LIN {X 0,Y 122.941,Z 954.134,A -85,B 0,C 180,E1 4520.76,E2 4520.76} C_VEL
LIN {X 0,Y 141.024,Z 945.626,A -85,B 0,C 180,E1 4515.408,E2 4515.408} C_VEL
LIN {X 0,Y 161.017,Z 934.73,A -85,B 0,C 180,E1 4511.199,E2 4511.199} C_VEL
LIN {X 0,Y 168.898,Z 929.93,A -85,B 0,C 180,E1 4509.837,E2 4509.837} C_VEL
LIN {X 0,Y 150.215,Z 939.451,A -85,B 0,C 180,E1 4506.112,E2 4506.112} C_VEL
LIN {X 0,Y 131.987,Z 947.261,A -85,B 0,C 180,E1 4501.242,E2 4501.242} C_VEL
LIN {X 0,Y 114.457,Z 953.373,A -85,B 0,C 180,E1 4494.654,E2 4494.654} C_VEL
LIN {X 0,Y 98.928,Z 957.725,A -85,B 0,C 180,E1 4485.934,E2 4485.934} C_VEL
LIN {X 0,Y 85.607,Z 960.518,A -85,B 0,C 180,E1 4473.649,E2 4473.649} C_VEL
LIN {X 0,Y 77.458,Z 961.489,A -85,B 0,C 180,E1 4459.579,E2 4459.579} C_VEL
LIN {X 0,Y 73.991,Z 961.027,A -85,B 0,C 180,E1 4445.504,E2 4445.504} C_VEL
LIN {X 0,Y 73.516,Z 959.727,A -85,B 0,C 180,E1 4432.349,E2 4432.349} C_VEL
LIN {X 0,Y 75.609,Z 957.116,A -85,B 0,C 180,E1 4418.348,E2 4418.348} C_VEL
LIN {X 0,Y 81.937,Z 952.659,A -85,B 0,C 180,E1 4403.68,E2 4403.68} C_VEL
LIN {X 0,Y 91.415,Z 946.902,A -85,B 0,C 180,E1 4392.153,E2 4392.153} C_VEL
LIN {X 0,Y 104.12,Z 938.983,A -85,B 0,C 180,E1 4382.54,E2 4382.54} C_VEL
LIN {X 0,Y 118.028,Z 929.614,A -85,B 0,C 180,E1 4375.407,E2 4375.407} C_VEL
LIN {X 0,Y 133.192,Z 918.259,A -85,B 0,C 180,E1 4369.779,E2 4369.779} C_VEL
LIN {X 0,Y 148.363,Z 905.384,A -85,B 0,C 180,E1 4365.492,E2 4365.492} C_VEL
LIN {X 0,Y 162.344,Z 891.921,A -85,B 0,C 180,E1 4362.339,E2 4362.339} C_VEL
LIN {X 0,Y 176.658,Z 876.08,A -85,B 0,C 180,E1 4359.661,E2 4359.661} C_VEL
LIN {X 0,Y 189.851,Z 859.095,A -85,B 0,C 180,E1 4357.561,E2 4357.561} C_VEL
LIN {X 0,Y 201.371,Z 841.861,A -85,B 0,C 180,E1 4355.961,E2 4355.961} C_VEL
LIN {X 0,Y 212.517,Z 822.257,A -85,B 0,C 180,E1 4354.571,E2 4354.571} C_VEL
LIN {X 0,Y 221.857,Z 802.538,A -85,B 0,C 180,E1 4353.507,E2 4353.507} C_VEL
LIN {X 0,Y 229.677,Z 782.335,A -85,B 0,C 180,E1 4352.672,E2 4352.672} C_VEL
LIN {X 0,Y 236.26,Z 760.464,A -85,B 0,C 180,E1 4351.999,E2 4351.999} C_VEL
LIN {X 0,Y 241.017,Z 738.583,A -85,B 0,C 180,E1 4351.512,E2 4351.512} C_VEL
LIN {X 0,Y 245.764,Z 704.393,A -85,B 0,C 180,E1 4350.967,E2 4350.967} C_VEL
LIN {X 0,Y 252.811,Z 648.458,A -85,B 0,C 180,E1 4350.086,E2 4350.086} C_VEL
LIN {X 0,Y 251.155,Z 644.335,A -85,B 0,C 180,E1 4346.898,E2 4346.898} C_VEL
LIN {X 0,Y 250.174,Z 641.772,A -85,B 0,C 180,E1 4344.31,E2 4344.31} C_VEL
LIN {X 0,Y 249.238,Z 639.151,A -85,B 0,C 180,E1 4340.152,E2 4340.152} C_VEL
LIN {X 0,Y 249.155,Z 638.957,A -85,B 0,C 180,E1 4334.645,E2 4334.645} C_VEL
LIN {X 0,Y 249.526,Z 639.799,A -85,B 0,C 180,E1 4332.262,E2 4332.262} C_VEL
LIN {X 0,Y 250.94,Z 643.145,A -85,B 0,C 180,E1 4327.787,E2 4327.787} C_VEL
LIN {X 0,Y 252.591,Z 647.143,A -85,B 0,C 180,E1 4324.428,E2 4324.428} C_VEL
LIN {X 0,Y 254.618,Z 652.06,A -85,B 0,C 180,E1 4321.288,E2 4321.288} C_VEL
LIN {X 0,Y 243.355,Z 742.447,A -85,B 0,C 180,E1 4319.848,E2 4319.848} C_VEL
LIN {X 0,Y 238.68,Z 764.766,A -85,B 0,C 180,E1 4319.412,E2 4319.412} C_VEL
LIN {X 0,Y 232.693,Z 785.189,A -85,B 0,C 180,E1 4318.95,E2 4318.95} C_VEL
LIN {X 0,Y 224.583,Z 806.826,A -85,B 0,C 180,E1 4318.285,E2 4318.285} C_VEL
LIN {X 0,Y 215.694,Z 826.159,A -85,B 0,C 180,E1 4317.468,E2 4317.468} C_VEL
LIN {X 0,Y 205.01,Z 845.556,A -85,B 0,C 180,E1 4316.366,E2 4316.366} C_VEL
LIN {X 0,Y 192.977,Z 863.966,A -85,B 0,C 180,E1 4314.948,E2 4314.948} C_VEL
LIN {X 0,Y 180.253,Z 880.755,A -85,B 0,C 180,E1 4313.213,E2 4313.213} C_VEL
LIN {X 0,Y 166.08,Z 897.05,A -85,B 0,C 180,E1 4310.907,E2 4310.907} C_VEL
LIN {X 0,Y 151.319,Z 911.904,A -85,B 0,C 180,E1 4307.969,E2 4307.969} C_VEL
LIN {X 0,Y 136.169,Z 925.263,A -85,B 0,C 180,E1 4304.161,E2 4304.161} C_VEL
LIN {X 0,Y 133.634,Z 927.346,A -85,B 0,C 180,E1 4303.421,E2 4303.421} C_VEL
LIN {X 0,Y 127.746,Z 931.563,A -85,B 0,C 180,E1 4302.123,E2 4302.123} C_VEL
LIN {X 0,Y 110.847,Z 941.115,A -85,B 0,C 180,E1 4299.58,E2 4299.58} C_VEL
LIN {X 0,Y 104.946,Z 944.656,A -85,B 0,C 180,E1 4297.699,E2 4297.699} C_VEL
LIN {X 0,Y 90.296,Z 953.759,A -85,B 0,C 180,E1 4289.381,E2 4289.381} C_VEL
LIN {X 0,Y 77.912,Z 961.092,A -85,B 0,C 180,E1 4278.122,E2 4278.122} C_VEL
LIN {X 0,Y 69.097,Z 966.731,A -85,B 0,C 180,E1 4263.378,E2 4263.378} C_VEL
LIN {X 0,Y 65.327,Z 970.268,A -85,B 0,C 180,E1 4247.844,E2 4247.844} C_VEL
LIN {X 0,Y 65.237,Z 972.242,A -85,B 0,C 180,E1 4233.533,E2 4233.533} C_VEL
LIN {X 0,Y 65.26,Z 972.617,A -85,B 0,C 180,E1 4227.384,E2 4227.384} C_VEL
LIN {X 0,Y 65.112,Z 972.66,A -85,B 0,C 180,E1 4213.057,E2 4213.057} C_VEL
LIN {X 0,Y 69.713,Z 971.183,A -85,B 0,C 180,E1 4194.833,E2 4194.833} C_VEL
LIN {X 0,Y 80.755,Z 967.951,A -85,B 0,C 180,E1 4178.764,E2 4178.764} C_VEL
LIN {X 0,Y 97.243,Z 962.683,A -85,B 0,C 180,E1 4166.583,E2 4166.583} C_VEL
LIN {X 0,Y 116.788,Z 955.393,A -85,B 0,C 180,E1 4158.178,E2 4158.178} C_VEL
LIN {X 0,Y 136.489,Z 946.767,A -85,B 0,C 180,E1 4152.694,E2 4152.694} C_VEL
LIN {X 0,Y 151.098,Z 939.539,A -85,B 0,C 180,E1 4149.665,E2 4149.665} C_VEL
LIN {X 0,Y 131.493,Z 947.642,A -85,B 0,C 180,E1 4145.181,E2 4145.181} C_VEL
LIN {X 0,Y 112.97,Z 953.837,A -85,B 0,C 180,E1 4139.187,E2 4139.187} C_VEL
LIN {X 0,Y 96.095,Z 958.284,A -85,B 0,C 180,E1 4131.019,E2 4131.019} C_VEL
LIN {X 0,Y 81.927,Z 961.07,A -85,B 0,C 180,E1 4119.958,E2 4119.958} C_VEL
LIN {X 0,Y 71.187,Z 962.264,A -85,B 0,C 180,E1 4104.52,E2 4104.52} C_VEL
LIN {X 0,Y 66.324,Z 961.804,A -85,B 0,C 180,E1 4088.152,E2 4088.152} C_VEL
LIN {X 0,Y 65.487,Z 960.535,A -85,B 0,C 180,E1 4073.633,E2 4073.633} C_VEL
LIN {X 0,Y 67.428,Z 958.096,A -85,B 0,C 180,E1 4058.509,E2 4058.509} C_VEL
LIN {X 0,Y 73.652,Z 954.042,A -85,B 0,C 180,E1 4042.966,E2 4042.966} C_VEL
LIN {X 0,Y 84.182,Z 948.085,A -85,B 0,C 180,E1 4029.837,E2 4029.837} C_VEL
LIN {X 0,Y 96.897,Z 940.726,A -85,B 0,C 180,E1 4020.297,E2 4020.297} C_VEL
LIN {X 0,Y 112.186,Z 931.095,A -85,B 0,C 180,E1 4012.683,E2 4012.683} C_VEL
LIN {X 0,Y 127.924,Z 919.921,A -85,B 0,C 180,E1 4007.146,E2 4007.146} C_VEL
LIN {X 0,Y 142.681,Z 908.045,A -85,B 0,C 180,E1 4003.204,E2 4003.204} C_VEL
LIN {X 0,Y 157.899,Z 893.971,A -85,B 0,C 180,E1 3999.976,E2 3999.976} C_VEL
LIN {X 0,Y 172.065,Z 878.845,A -85,B 0,C 180,E1 3997.506,E2 3997.506} C_VEL
LIN {X 0,Y 185.501,Z 862.283,A -85,B 0,C 180,E1 3995.513,E2 3995.513} C_VEL
LIN {X 0,Y 198.155,Z 844.091,A -85,B 0,C 180,E1 3993.889,E2 3993.889} C_VEL
LIN {X 0,Y 209.006,Z 825.752,A -85,B 0,C 180,E1 3992.644,E2 3992.644} C_VEL
LIN {X 0,Y 218.958,Z 805.636,A -85,B 0,C 180,E1 3991.602,E2 3991.602} C_VEL
LIN {X 0,Y 227.293,Z 784.765,A -85,B 0,C 180,E1 3990.783,E2 3990.783} C_VEL
LIN {X 0,Y 233.847,Z 763.8,A -85,B 0,C 180,E1 3990.168,E2 3990.168} C_VEL
LIN {X 0,Y 238.893,Z 742.056,A -85,B 0,C 180,E1 3989.697,E2 3989.697} C_VEL
LIN {X 0,Y 243.144,Z 713.786,A -85,B 0,C 180,E1 3989.258,E2 3989.258} C_VEL
LIN {X 0,Y 250.728,Z 654.36,A -85,B 0,C 180,E1 3988.374,E2 3988.374} C_VEL
LIN {X 0,Y 249.208,Z 650.025,A -85,B 0,C 180,E1 3984.663,E2 3984.663} C_VEL
LIN {X 0,Y 248.14,Z 647.059,A -85,B 0,C 180,E1 3980.03,E2 3980.03} C_VEL
LIN {X 0,Y 248.104,Z 646.928,A -85,B 0,C 180,E1 3974.47,E2 3974.47} C_VEL
LIN {X 0,Y 248.426,Z 647.784,A -85,B 0,C 180,E1 3972.317,E2 3972.317} C_VEL
LIN {X 0,Y 249.675,Z 650.864,A -85,B 0,C 180,E1 3968.174,E2 3968.174} C_VEL
LIN {X 0,Y 251.255,Z 654.891,A -85,B 0,C 180,E1 3964.794,E2 3964.794} C_VEL
LIN {X 0,Y 252.333,Z 657.73,A -85,B 0,C 180,E1 3962.976,E2 3962.976} C_VEL
LIN {X 0,Y 241.585,Z 742.196,A -85,B 0,C 180,E1 3961.695,E2 3961.695} C_VEL
LIN {X 0,Y 236.821,Z 764.595,A -85,B 0,C 180,E1 3961.289,E2 3961.289} C_VEL
LIN {X 0,Y 230.507,Z 785.745,A -85,B 0,C 180,E1 3960.853,E2 3960.853} C_VEL
LIN {X 0,Y 222.409,Z 806.917,A -85,B 0,C 180,E1 3960.258,E2 3960.258} C_VEL
LIN {X 0,Y 212.993,Z 826.926,A -85,B 0,C 180,E1 3959.48,E2 3959.48} C_VEL
LIN {X 0,Y 202.059,Z 846.323,A -85,B 0,C 180,E1 3958.458,E2 3958.458} C_VEL
LIN {X 0,Y 189.725,Z 864.773,A -85,B 0,C 180,E1 3957.137,E2 3957.137} C_VEL
LIN {X 0,Y 176.536,Z 881.669,A -85,B 0,C 180,E1 3955.496,E2 3955.496} C_VEL
LIN {X 0,Y 162.089,Z 897.747,A -85,B 0,C 180,E1 3953.335,E2 3953.335} C_VEL
LIN {X 0,Y 146.987,Z 912.405,A -85,B 0,C 180,E1 3950.56,E2 3950.56} C_VEL
LIN {X 0,Y 131.407,Z 925.655,A -85,B 0,C 180,E1 3946.923,E2 3946.923} C_VEL
LIN {X 0,Y 115.629,Z 937.38,A -85,B 0,C 180,E1 3942.052,E2 3942.052} C_VEL
LIN {X 0,Y 104.946,Z 944.656,A -85,B 0,C 180,E1 3937.699,E2 3937.699} C_VEL
LIN {X 0,Y 99.077,Z 948.011,A -85,B 0,C 180,E1 3935.556,E2 3935.556} C_VEL
LIN {X 0,Y 81.245,Z 955.584,A -85,B 0,C 180,E1 3929.929,E2 3929.929} C_VEL
LIN {X 0,Y 76.561,Z 957.802,A -85,B 0,C 180,E1 3926.89,E2 3926.89} C_VEL
LIN {X 0,Y 65.424,Z 963.843,A -85,B 0,C 180,E1 3913.474,E2 3913.474} C_VEL
LIN {X 0,Y 58.448,Z 968.456,A -85,B 0,C 180,E1 3895.342,E2 3895.342} C_VEL
LIN {X 0,Y 57.026,Z 970.951,A -85,B 0,C 180,E1 3878.085,E2 3878.085} C_VEL
LIN {X 0,Y 57.431,Z 971.671,A -85,B 0,C 180,E1 3870.021,E2 3870.021} C_VEL
LIN {X 0,Y 56.913,Z 971.987,A -85,B 0,C 180,E1 3857.852,E2 3857.852} C_VEL
LIN {X 0,Y 60.005,Z 971.266,A -85,B 0,C 180,E1 3838.185,E2 3838.185} C_VEL
LIN {X 0,Y 70.752,Z 968.681,A -85,B 0,C 180,E1 3819.02,E2 3819.02} C_VEL
LIN {X 0,Y 86.659,Z 964.409,A -85,B 0,C 180,E1 3805.884,E2 3805.884} C_VEL
LIN {X 0,Y 105.789,Z 958.337,A -85,B 0,C 180,E1 3797.036,E2 3797.036} C_VEL
LIN {X 0,Y 126.327,Z 950.451,A -85,B 0,C 180,E1 3791.115,E2 3791.115} C_VEL
LIN {X 0,Y 133.3,Z 947.425,A -85,B 0,C 180,E1 3789.497,E2 3789.497} C_VEL
LIN {X 0,Y 112.982,Z 954.102,A -85,B 0,C 180,E1 3784.058,E2 3784.058} C_VEL
LIN {X 0,Y 94.015,Z 958.884,A -85,B 0,C 180,E1 3776.34,E2 3776.34} C_VEL
LIN {X 0,Y 77.524,Z 961.836,A -85,B 0,C 180,E1 3765.241,E2 3765.241} C_VEL
LIN {X 0,Y 65.004,Z 963.029,A -85,B 0,C 180,E1 3749.43,E2 3749.43} C_VEL
LIN {X 0,Y 58.82,Z 962.581,A -85,B 0,C 180,E1 3731.496,E2 3731.496} C_VEL
LIN {X 0,Y 57.477,Z 961.326,A -85,B 0,C 180,E1 3715.225,E2 3715.225} C_VEL
LIN {X 0,Y 59.506,Z 958.849,A -85,B 0,C 180,E1 3697.52,E2 3697.52} C_VEL
LIN {X 0,Y 66.296,Z 954.862,A -85,B 0,C 180,E1 3680.432,E2 3680.432} C_VEL
LIN {X 0,Y 77.764,Z 948.921,A -85,B 0,C 180,E1 3666.494,E2 3666.494} C_VEL
LIN {X 0,Y 91.366,Z 941.604,A -85,B 0,C 180,E1 3656.812,E2 3656.812} C_VEL
LIN {X 0,Y 107.459,Z 932.02,A -85,B 0,C 180,E1 3649.345,E2 3649.345} C_VEL
LIN {X 0,Y 123.463,Z 921.171,A -85,B 0,C 180,E1 3644.146,E2 3644.146} C_VEL
LIN {X 0,Y 139.051,Z 909.084,A -85,B 0,C 180,E1 3640.33,E2 3640.33} C_VEL
LIN {X 0,Y 154.659,Z 895.043,A -85,B 0,C 180,E1 3637.317,E2 3637.317} C_VEL
LIN {X 0,Y 168.722,Z 880.448,A -85,B 0,C 180,E1 3635.089,E2 3635.089} C_VEL
LIN {X 0,Y 182.82,Z 863.531,A -85,B 0,C 180,E1 3633.19,E2 3633.19} C_VEL
LIN {X 0,Y 195.204,Z 846.205,A -85,B 0,C 180,E1 3631.75,E2 3631.75} C_VEL
LIN {X 0,Y 206.692,Z 827.288,A -85,B 0,C 180,E1 3630.555,E2 3630.555} C_VEL
LIN {X 0,Y 216.775,Z 807.316,A -85,B 0,C 180,E1 3629.598,E2 3629.598} C_VEL
LIN {X 0,Y 224.941,Z 787.416,A -85,B 0,C 180,E1 3628.869,E2 3628.869} C_VEL
LIN {X 0,Y 231.868,Z 766.149,A -85,B 0,C 180,E1 3628.28,E2 3628.28} C_VEL
LIN {X 0,Y 237.323,Z 743.515,A -85,B 0,C 180,E1 3627.821,E2 3627.821} C_VEL
LIN {X 0,Y 241.195,Z 719.145,A -85,B 0,C 180,E1 3627.462,E2 3627.462} C_VEL
LIN {X 0,Y 248.821,Z 660.307,A -85,B 0,C 180,E1 3626.652,E2 3626.652} C_VEL
LIN {X 0,Y 247.741,Z 657.272,A -85,B 0,C 180,E1 3623.551,E2 3623.551} C_VEL
LIN {X 0,Y 247.039,Z 654.961,A -85,B 0,C 180,E1 3619.876,E2 3619.876} C_VEL
LIN {X 0,Y 247.02,Z 654.849,A -85,B 0,C 180,E1 3614.535,E2 3614.535} C_VEL
LIN {X 0,Y 247.327,Z 655.766,A -85,B 0,C 180,E1 3612.373,E2 3612.373} C_VEL
LIN {X 0,Y 248.463,Z 658.715,A -85,B 0,C 180,E1 3608.447,E2 3608.447} C_VEL
LIN {X 0,Y 249.966,Z 662.73,A -85,B 0,C 180,E1 3605.096,E2 3605.096} C_VEL
LIN {X 0,Y 250.168,Z 663.427,A -85,B 0,C 180,E1 3604.689,E2 3604.689} C_VEL
LIN {X 0,Y 240.027,Z 741.859,A -85,B 0,C 180,E1 3603.566,E2 3603.566} C_VEL
LIN {X 0,Y 235.208,Z 764.284,A -85,B 0,C 180,E1 3603.192,E2 3603.192} C_VEL
LIN {X 0,Y 228.755,Z 785.662,A -85,B 0,C 180,E1 3602.801,E2 3602.801} C_VEL
LIN {X 0,Y 220.844,Z 806.154,A -85,B 0,C 180,E1 3602.292,E2 3602.292} C_VEL
LIN {X 0,Y 211.644,Z 825.647,A -85,B 0,C 180,E1 3601.625,E2 3601.625} C_VEL
LIN {X 0,Y 200.502,Z 845.307,A -85,B 0,C 180,E1 3600.708,E2 3600.708} C_VEL
LIN {X 0,Y 187.995,Z 863.798,A -85,B 0,C 180,E1 3599.526,E2 3599.526} C_VEL
LIN {X 0,Y 175.086,Z 880.175,A -85,B 0,C 180,E1 3598.107,E2 3598.107} C_VEL
LIN {X 0,Y 160.352,Z 896.398,A -85,B 0,C 180,E1 3596.167,E2 3596.167} C_VEL
LIN {X 0,Y 145.842,Z 910.358,A -85,B 0,C 180,E1 3593.827,E2 3593.827} C_VEL
LIN {X 0,Y 129.76,Z 923.761,A -85,B 0,C 180,E1 3590.551,E2 3590.551} C_VEL
LIN {X 0,Y 113.948,Z 935.294,A -85,B 0,C 180,E1 3586.297,E2 3586.297} C_VEL
LIN {X 0,Y 96.937,Z 946.232,A -85,B 0,C 180,E1 3579.853,E2 3579.853} C_VEL
LIN {X 0,Y 82.081,Z 954.798,A -85,B 0,C 180,E1 3571.317,E2 3571.317} C_VEL
LIN {X 0,Y 76.561,Z 957.802,A -85,B 0,C 180,E1 3566.89,E2 3566.89} C_VEL
LIN {X 0,Y 71.268,Z 960.225,A -85,B 0,C 180,E1 3562.908,E2 3562.908} C_VEL
LIN {X 0,Y 55.416,Z 965.293,A -85,B 0,C 180,E1 3549.962,E2 3549.962} C_VEL
LIN {X 0,Y 52.571,Z 966.514,A -85,B 0,C 180,E1 3544.351,E2 3544.351} C_VEL
LIN {X 0,Y 49.05,Z 969.709,A -85,B 0,C 180,E1 3522.983,E2 3522.983} C_VEL
LIN {X 0,Y 49.46,Z 970.859,A -85,B 0,C 180,E1 3510.025,E2 3510.025} C_VEL
LIN {X 0,Y 49.106,Z 971.19,A -85,B 0,C 180,E1 3493.464,E2 3493.464} C_VEL
LIN {X 0,Y 54.103,Z 970.401,A -85,B 0,C 180,E1 3471.103,E2 3471.103} C_VEL
LIN {X 0,Y 67.203,Z 967.806,A -85,B 0,C 180,E1 3452.036,E2 3452.036} C_VEL
LIN {X 0,Y 85.869,Z 963.286,A -85,B 0,C 180,E1 3439.458,E2 3439.458} C_VEL
LIN {X 0,Y 106.229,Z 957.201,A -85,B 0,C 180,E1 3431.863,E2 3431.863} C_VEL
LIN {X 0,Y 115.656,Z 953.892,A -85,B 0,C 180,E1 3429.36,E2 3429.36} C_VEL
LIN {X 0,Y 95.075,Z 959.065,A -85,B 0,C 180,E1 3422.787,E2 3422.787} C_VEL
LIN {X 0,Y 76.527,Z 962.262,A -85,B 0,C 180,E1 3413.055,E2 3413.055} C_VEL
LIN {X 0,Y 62.013,Z 963.646,A -85,B 0,C 180,E1 3399.193,E2 3399.193} C_VEL
LIN {X 0,Y 52.173,Z 963.481,A -85,B 0,C 180,E1 3378.329,E2 3378.329} C_VEL
LIN {X 0,Y 49.565,Z 962.31,A -85,B 0,C 180,E1 3359.833,E2 3359.833} C_VEL
LIN {X 0,Y 50.826,Z 960.22,A -85,B 0,C 180,E1 3340.173,E2 3340.173} C_VEL
LIN {X 0,Y 57.078,Z 956.585,A -85,B 0,C 180,E1 3320.908,E2 3320.908} C_VEL
LIN {X 0,Y 68.867,Z 951.03,A -85,B 0,C 180,E1 3305.081,E2 3305.081} C_VEL
LIN {X 0,Y 82.999,Z 944.158,A -85,B 0,C 180,E1 3294.657,E2 3294.657} C_VEL
LIN {X 0,Y 98.79,Z 935.543,A -85,B 0,C 180,E1 3287.289,E2 3287.289} C_VEL
LIN {X 0,Y 114.757,Z 925.504,A -85,B 0,C 180,E1 3282.138,E2 3282.138} C_VEL
LIN {X 0,Y 131.136,Z 913.677,A -85,B 0,C 180,E1 3278.236,E2 3278.236} C_VEL
LIN {X 0,Y 147.132,Z 900.325,A -85,B 0,C 180,E1 3275.285,E2 3275.285} C_VEL
LIN {X 0,Y 162.227,Z 885.765,A -85,B 0,C 180,E1 3273.037,E2 3273.037} C_VEL
LIN {X 0,Y 176.604,Z 869.569,A -85,B 0,C 180,E1 3271.241,E2 3271.241} C_VEL
LIN {X 0,Y 189.542,Z 852.545,A -85,B 0,C 180,E1 3269.844,E2 3269.844} C_VEL
LIN {X 0,Y 201.74,Z 833.693,A -85,B 0,C 180,E1 3268.679,E2 3268.679} C_VEL
LIN {X 0,Y 212.427,Z 813.966,A -85,B 0,C 180,E1 3267.754,E2 3267.754} C_VEL
LIN {X 0,Y 221.179,Z 794.421,A -85,B 0,C 180,E1 3267.049,E2 3267.049} C_VEL
LIN {X 0,Y 228.712,Z 773.36,A -85,B 0,C 180,E1 3266.47,E2 3266.47} C_VEL
LIN {X 0,Y 234.617,Z 751.43,A -85,B 0,C 180,E1 3266.024,E2 3266.024} C_VEL
LIN {X 0,Y 238.698,Z 729.638,A -85,B 0,C 180,E1 3265.704,E2 3265.704} C_VEL
LIN {X 0,Y 247.05,Z 666.591,A -85,B 0,C 180,E1 3264.893,E2 3264.893} C_VEL
LIN {X 0,Y 246.332,Z 664.418,A -85,B 0,C 180,E1 3262.255,E2 3262.255} C_VEL
LIN {X 0,Y 245.91,Z 662.815,A -85,B 0,C 180,E1 3259.476,E2 3259.476} C_VEL
LIN {X 0,Y 245.969,Z 662.824,A -85,B 0,C 180,E1 3254.358,E2 3254.358} C_VEL
LIN {X 0,Y 246.325,Z 664.07,A -85,B 0,C 180,E1 3251.948,E2 3251.948} C_VEL
LIN {X 0,Y 247.259,Z 666.566,A -85,B 0,C 180,E1 3248.723,E2 3248.723} C_VEL
LIN {X 0,Y 248.197,Z 669.297,A -85,B 0,C 180,E1 3246.428,E2 3246.428} C_VEL
LIN {X 0,Y 238.688,Z 741.456,A -85,B 0,C 180,E1 3245.459,E2 3245.459} C_VEL
LIN {X 0,Y 233.814,Z 763.887,A -85,B 0,C 180,E1 3245.119,E2 3245.119} C_VEL
LIN {X 0,Y 227.322,Z 785.215,A -85,B 0,C 180,E1 3244.78,E2 3244.78} C_VEL
LIN {X 0,Y 219.108,Z 806.245,A -85,B 0,C 180,E1 3244.326,E2 3244.326} C_VEL
LIN {X 0,Y 209.425,Z 826.352,A -85,B 0,C 180,E1 3243.717,E2 3243.717} C_VEL
LIN {X 0,Y 198.243,Z 845.688,A -85,B 0,C 180,E1 3242.914,E2 3242.914} C_VEL
LIN {X 0,Y 185.468,Z 864.286,A -85,B 0,C 180,E1 3241.855,E2 3241.855} C_VEL
LIN {X 0,Y 171.999,Z 880.964,A -85,B 0,C 180,E1 3240.551,E2 3240.551} C_VEL
LIN {X 0,Y 157.028,Z 896.988,A -85,B 0,C 180,E1 3238.801,E2 3238.801} C_VEL
LIN {X 0,Y 141.258,Z 911.595,A -85,B 0,C 180,E1 3236.518,E2 3236.518} C_VEL
LIN {X 0,Y 124.811,Z 924.796,A -85,B 0,C 180,E1 3233.466,E2 3233.466} C_VEL
LIN {X 0,Y 106.973,Z 937.101,A -85,B 0,C 180,E1 3228.987,E2 3228.987} C_VEL
LIN {X 0,Y 90.887,Z 946.713,A -85,B 0,C 180,E1 3223.197,E2 3223.197} C_VEL
LIN {X 0,Y 74.511,Z 955.408,A -85,B 0,C 180,E1 3214.07,E2 3214.07} C_VEL
LIN {X 0,Y 60.823,Z 962.168,A -85,B 0,C 180,E1 3200.619,E2 3200.619} C_VEL
LIN {X 0,Y 52.571,Z 966.514,A -85,B 0,C 180,E1 3184.351,E2 3184.351} C_VEL
LIN {X 0,Y 49.652,Z 967.94,A -85,B 0,C 180,E1 3176.39,E2 3176.39} C_VEL
LIN {X 0,Y 45.336,Z 969.237,A -85,B 0,C 180,E1 3164.722,E2 3164.722} C_VEL
LIN {X 0,Y 41.036,Z 970.251,A -85,B 0,C 180,E1 3141.827,E2 3141.827} C_VEL
LIN {X 0,Y 44.01,Z 970.224,A -85,B 0,C 180,E1 3115.426,E2 3115.426} C_VEL
LIN {X 0,Y 56.367,Z 968.429,A -85,B 0,C 180,E1 3092.147,E2 3092.147} C_VEL
LIN {X 0,Y 75.529,Z 964.711,A -85,B 0,C 180,E1 3077.668,E2 3077.668} C_VEL
LIN {X 0,Y 97.263,Z 959.178,A -85,B 0,C 180,E1 3069.381,E2 3069.381} C_VEL
LIN {X 0,Y 97.673,Z 959.038,A -85,B 0,C 180,E1 3069.134,E2 3069.134} C_VEL
LIN {X 0,Y 77.99,Z 962.496,A -85,B 0,C 180,E1 3061.456,E2 3061.456} C_VEL
LIN {X 0,Y 60.106,Z 964.319,A -85,B 0,C 180,E1 3048.836,E2 3048.836} C_VEL
LIN {X 0,Y 46.928,Z 964.45,A -85,B 0,C 180,E1 3028.405,E2 3028.405} C_VEL
LIN {X 0,Y 41.863,Z 963.217,A -85,B 0,C 180,E1 3004.938,E2 3004.938} C_VEL
LIN {X 0,Y 42.053,Z 961.569,A -85,B 0,C 180,E1 2985.131,E2 2985.131} C_VEL
LIN {X 0,Y 47.821,Z 958.273,A -85,B 0,C 180,E1 2961.559,E2 2961.559} C_VEL
LIN {X 0,Y 59.3,Z 953.426,A -85,B 0,C 180,E1 2943.977,E2 2943.977} C_VEL
LIN {X 0,Y 74.981,Z 946.454,A -85,B 0,C 180,E1 2931.886,E2 2931.886} C_VEL
LIN {X 0,Y 91.554,Z 938.084,A -85,B 0,C 180,E1 2924.345,E2 2924.345} C_VEL
LIN {X 0,Y 109.353,Z 927.631,A -85,B 0,C 180,E1 2918.981,E2 2918.981} C_VEL
LIN {X 0,Y 126.252,Z 916.05,A -85,B 0,C 180,E1 2915.328,E2 2915.328} C_VEL
LIN {X 0,Y 142.494,Z 903.111,A -85,B 0,C 180,E1 2912.633,E2 2912.633} C_VEL
LIN {X 0,Y 157.945,Z 888.703,A -85,B 0,C 180,E1 2910.566,E2 2910.566} C_VEL
LIN {X 0,Y 172.538,Z 872.912,A -85,B 0,C 180,E1 2908.938,E2 2908.938} C_VEL
LIN {X 0,Y 186.712,Z 854.951,A -85,B 0,C 180,E1 2907.582,E2 2907.582} C_VEL
LIN {X 0,Y 198.976,Z 836.61,A -85,B 0,C 180,E1 2906.551,E2 2906.551} C_VEL
LIN {X 0,Y 209.783,Z 817.41,A -85,B 0,C 180,E1 2905.726,E2 2905.726} C_VEL
LIN {X 0,Y 219.116,Z 797.237,A -85,B 0,C 180,E1 2905.061,E2 2905.061} C_VEL
LIN {X 0,Y 226.721,Z 776.656,A -85,B 0,C 180,E1 2904.544,E2 2904.544} C_VEL
LIN {X 0,Y 232.87,Z 755.049,A -85,B 0,C 180,E1 2904.134,E2 2904.134} C_VEL
LIN {X 0,Y 237.489,Z 731.912,A -85,B 0,C 180,E1 2903.817,E2 2903.817} C_VEL
LIN {X 0,Y 245.425,Z 672.981,A -85,B 0,C 180,E1 2903.087,E2 2903.087} C_VEL
LIN {X 0,Y 244.815,Z 670.719,A -85,B 0,C 180,E1 2899.319,E2 2899.319} C_VEL
LIN {X 0,Y 244.915,Z 670.798,A -85,B 0,C 180,E1 2894.179,E2 2894.179} C_VEL
LIN {X 0,Y 245.954,Z 674.02,A -85,B 0,C 180,E1 2889.359,E2 2889.359} C_VEL
LIN {X 0,Y 246.326,Z 675.457,A -85,B 0,C 180,E1 2888.187,E2 2888.187} C_VEL
LIN {X 0,Y 237.52,Z 741.248,A -85,B 0,C 180,E1 2887.366,E2 2887.366} C_VEL
LIN {X 0,Y 232.622,Z 763.586,A -85,B 0,C 180,E1 2887.064,E2 2887.064} C_VEL
LIN {X 0,Y 226.27,Z 784.353,A -85,B 0,C 180,E1 2886.786,E2 2886.786} C_VEL
LIN {X 0,Y 218.355,Z 804.674,A -85,B 0,C 180,E1 2886.425,E2 2886.425} C_VEL
LIN {X 0,Y 209.109,Z 824.072,A -85,B 0,C 180,E1 2885.943,E2 2885.943} C_VEL
LIN {X 0,Y 197.822,Z 843.695,A -85,B 0,C 180,E1 2885.267,E2 2885.267} C_VEL
LIN {X 0,Y 185.541,Z 861.582,A -85,B 0,C 180,E1 2884.419,E2 2884.419} C_VEL
LIN {X 0,Y 172.094,Z 878.388,A -85,B 0,C 180,E1 2883.332,E2 2883.332} C_VEL
LIN {X 0,Y 157.078,Z 894.547,A -85,B 0,C 180,E1 2881.874,E2 2881.874} C_VEL
LIN {X 0,Y 141.475,Z 909.058,A -85,B 0,C 180,E1 2880.001,E2 2880.001} C_VEL
LIN {X 0,Y 125.118,Z 922.093,A -85,B 0,C 180,E1 2877.508,E2 2877.508} C_VEL
LIN {X 0,Y 108.566,Z 933.528,A -85,B 0,C 180,E1 2874.16,E2 2874.16} C_VEL
LIN {X 0,Y 91.327,Z 943.859,A -85,B 0,C 180,E1 2869.275,E2 2869.275} C_VEL
LIN {X 0,Y 74.535,Z 952.576,A -85,B 0,C 180,E1 2862.031,E2 2862.031} C_VEL
LIN {X 0,Y 58.725,Z 959.756,A -85,B 0,C 180,E1 2850.305,E2 2850.305} C_VEL
LIN {X 0,Y 46.61,Z 965.152,A -85,B 0,C 180,E1 2831.716,E2 2831.716} C_VEL
LIN {X 0,Y 41.238,Z 968.686,A -85,B 0,C 180,E1 2806.945,E2 2806.945} C_VEL
LIN {X 0,Y 41.483,Z 970.04,A -85,B 0,C 180,E1 2790.029,E2 2790.029} C_VEL
LIN {X 0,Y 41.036,Z 970.251,A -85,B 0,C 180,E1 2781.827,E2 2781.827} C_VEL
LIN {X 0,Y 40.4,Z 970.355,A -85,B 0,C 180,E1 2771.731,E2 2771.731} C_VEL
LIN {X 0,Y 39.592,Z 969.827,A -85,B 0,C 180,E1 2754.072,E2 2754.072} C_VEL
LIN {X 0,Y 42.141,Z 969.096,A -85,B 0,C 180,E1 2738.673,E2 2738.673} C_VEL
LIN {X 0,Y 44.915,Z 968.741,A -85,B 0,C 180,E1 2733.145,E2 2733.145} C_VEL
LIN {X 0,Y 63.519,Z 966.077,A -85,B 0,C 180,E1 2716.293,E2 2716.293} C_VEL
LIN {X 0,Y 79.946,Z 962.887,A -85,B 0,C 180,E1 2708.986,E2 2708.986} C_VEL
LIN {X 0,Y 59.98,Z 964.975,A -85,B 0,C 180,E1 2698.847,E2 2698.847} C_VEL
LIN {X 0,Y 43.414,Z 965.282,A -85,B 0,C 180,E1 2680.689,E2 2680.689} C_VEL
LIN {X 0,Y 34.491,Z 964.096,A -85,B 0,C 180,E1 2651.767,E2 2651.767} C_VEL
LIN {X 0,Y 33.836,Z 962.469,A -85,B 0,C 180,E1 2627.149,E2 2627.149} C_VEL
LIN {X 0,Y 39.513,Z 959.502,A -85,B 0,C 180,E1 2599.766,E2 2599.766} C_VEL
LIN {X 0,Y 52.029,Z 954.721,A -85,B 0,C 180,E1 2579.865,E2 2579.865} C_VEL
LIN {X 0,Y 68.44,Z 948.095,A -85,B 0,C 180,E1 2567.754,E2 2567.754} C_VEL
LIN {X 0,Y 86.797,Z 939.458,A -85,B 0,C 180,E1 2560.175,E2 2560.175} C_VEL
LIN {X 0,Y 104.4,Z 929.676,A -85,B 0,C 180,E1 2555.488,E2 2555.488} C_VEL
LIN {X 0,Y 122.325,Z 917.935,A -85,B 0,C 180,E1 2552.095,E2 2552.095} C_VEL
LIN {X 0,Y 139.576,Z 904.559,A -85,B 0,C 180,E1 2549.624,E2 2549.624} C_VEL
LIN {X 0,Y 154.954,Z 890.624,A -85,B 0,C 180,E1 2547.857,E2 2547.857} C_VEL
LIN {X 0,Y 170.245,Z 874.523,A -85,B 0,C 180,E1 2546.396,E2 2546.396} C_VEL
LIN {X 0,Y 184.096,Z 857.442,A -85,B 0,C 180,E1 2545.26,E2 2545.26} C_VEL
LIN {X 0,Y 196.494,Z 839.499,A -85,B 0,C 180,E1 2544.367,E2 2544.367} C_VEL
LIN {X 0,Y 207.768,Z 819.984,A -85,B 0,C 180,E1 2543.625,E2 2543.625} C_VEL
LIN {X 0,Y 217.317,Z 799.897,A -85,B 0,C 180,E1 2543.037,E2 2543.037} C_VEL
LIN {X 0,Y 225.239,Z 779.219,A -85,B 0,C 180,E1 2542.572,E2 2542.572} C_VEL
LIN {X 0,Y 231.814,Z 756.881,A -85,B 0,C 180,E1 2542.193,E2 2542.193} C_VEL
LIN {X 0,Y 236.388,Z 735.072,A -85,B 0,C 180,E1 2541.922,E2 2541.922} C_VEL
LIN {X 0,Y 243.972,Z 679.848,A -85,B 0,C 180,E1 2541.348,E2 2541.348} C_VEL
LIN {X 0,Y 243.721,Z 678.624,A -85,B 0,C 180,E1 2539.16,E2 2539.16} C_VEL
LIN {X 0,Y 243.83,Z 678.72,A -85,B 0,C 180,E1 2534.244,E2 2534.244} C_VEL
LIN {X 0,Y 244.676,Z 681.539,A -85,B 0,C 180,E1 2529.972,E2 2529.972} C_VEL
LIN {X 0,Y 236.547,Z 741.099,A -85,B 0,C 180,E1 2529.287,E2 2529.287} C_VEL
LIN {X 0,Y 231.598,Z 763.418,A -85,B 0,C 180,E1 2529.024,E2 2529.024} C_VEL
LIN {X 0,Y 225.131,Z 784.341,A -85,B 0,C 180,E1 2528.796,E2 2528.796} C_VEL
LIN {X 0,Y 217.061,Z 804.805,A -85,B 0,C 180,E1 2528.503,E2 2528.503} C_VEL
LIN {X 0,Y 207.557,Z 824.434,A -85,B 0,C 180,E1 2528.101,E2 2528.101} C_VEL
LIN {X 0,Y 196.117,Z 844.05,A -85,B 0,C 180,E1 2527.54,E2 2527.54} C_VEL
LIN {X 0,Y 183.282,Z 862.456,A -85,B 0,C 180,E1 2526.808,E2 2526.808} C_VEL
LIN {X 0,Y 169.382,Z 879.414,A -85,B 0,C 180,E1 2525.875,E2 2525.875} C_VEL
LIN {X 0,Y 153.995,Z 895.52,A -85,B 0,C 180,E1 2524.621,E2 2524.621} C_VEL
LIN {X 0,Y 138.189,Z 909.777,A -85,B 0,C 180,E1 2523.02,E2 2523.02} C_VEL
LIN {X 0,Y 121.012,Z 923.08,A -85,B 0,C 180,E1 2520.786,E2 2520.786} C_VEL
LIN {X 0,Y 103.092,Z 934.839,A -85,B 0,C 180,E1 2517.628,E2 2517.628} C_VEL
LIN {X 0,Y 85.607,Z 944.647,A -85,B 0,C 180,E1 2513.211,E2 2513.211} C_VEL
LIN {X 0,Y 67.958,Z 953.127,A -85,B 0,C 180,E1 2506.249,E2 2506.249} C_VEL
LIN {X 0,Y 51.108,Z 960.135,A -85,B 0,C 180,E1 2494.201,E2 2494.201} C_VEL
LIN {X 0,Y 38.122,Z 965.193,A -85,B 0,C 180,E1 2473.036,E2 2473.036} C_VEL
LIN {X 0,Y 33.096,Z 968.375,A -85,B 0,C 180,E1 2442.246,E2 2442.246} C_VEL
LIN {X 0,Y 33.499,Z 969.174,A -85,B 0,C 180,E1 2430.036,E2 2430.036} C_VEL
LIN {X 0,Y 34.491,Z 969.593,A -85,B 0,C 180,E1 2400.516,E2 2400.516} C_VEL
LIN {X 0,Y 44.915,Z 968.741,A -85,B 0,C 180,E1 2373.145,E2 2373.145} C_VEL
LIN {X 0,Y 47.728,Z 968.342,A -85,B 0,C 180,E1 2367.707,E2 2367.707} C_VEL
LIN {X 0,Y 54.478,Z 966.757,A -85,B 0,C 180,E1 2353.392,E2 2353.392} C_VEL
LIN {X 0,Y 57.979,Z 966.129,A -85,B 0,C 180,E1 2350.587,E2 2350.587} C_VEL
LIN {X 0,Y 61.833,Z 965.506,A -85,B 0,C 180,E1 2348.721,E2 2348.721} C_VEL
LIN {X 0,Y 42.167,Z 966.114,A -85,B 0,C 180,E1 2334.481,E2 2334.481} C_VEL
LIN {X 0,Y 28.604,Z 965.173,A -85,B 0,C 180,E1 2305.987,E2 2305.987} C_VEL
LIN {X 0,Y 25.58,Z 963.514,A -85,B 0,C 180,E1 2272.956,E2 2272.956} C_VEL
LIN {X 0,Y 29.617,Z 961.201,A -85,B 0,C 180,E1 2242.198,E2 2242.198} C_VEL
LIN {X 0,Y 43.288,Z 956.604,A -85,B 0,C 180,E1 2216.302,E2 2216.302} C_VEL
LIN {X 0,Y 59.82,Z 950.735,A -85,B 0,C 180,E1 2204.023,E2 2204.023} C_VEL
LIN {X 0,Y 78.818,Z 942.625,A -85,B 0,C 180,E1 2196.603,E2 2196.603} C_VEL
LIN {X 0,Y 96.935,Z 933.27,A -85,B 0,C 180,E1 2192.221,E2 2192.221} C_VEL
LIN {X 0,Y 114.667,Z 922.439,A -85,B 0,C 180,E1 2189.231,E2 2189.231} C_VEL
LIN {X 0,Y 131.981,Z 910.008,A -85,B 0,C 180,E1 2187.037,E2 2187.037} C_VEL
LIN {X 0,Y 148.341,Z 896.264,A -85,B 0,C 180,E1 2185.403,E2 2185.403} C_VEL
LIN {X 0,Y 164.299,Z 880.456,A -85,B 0,C 180,E1 2184.085,E2 2184.085} C_VEL
LIN {X 0,Y 178.554,Z 863.891,A -85,B 0,C 180,E1 2183.079,E2 2183.079} C_VEL
LIN {X 0,Y 191.79,Z 845.826,A -85,B 0,C 180,E1 2182.265,E2 2182.265} C_VEL
LIN {X 0,Y 203.701,Z 826.515,A -85,B 0,C 180,E1 2181.602,E2 2181.602} C_VEL
LIN {X 0,Y 213.298,Z 807.959,A -85,B 0,C 180,E1 2181.108,E2 2181.108} C_VEL
LIN {X 0,Y 222.284,Z 786.455,A -85,B 0,C 180,E1 2180.663,E2 2180.663} C_VEL
LIN {X 0,Y 229.167,Z 765.248,A -85,B 0,C 180,E1 2180.331,E2 2180.331} C_VEL
LIN {X 0,Y 234.371,Z 743.594,A -85,B 0,C 180,E1 2180.07,E2 2180.07} C_VEL
LIN {X 0,Y 238.874,Z 714.846,A -85,B 0,C 180,E1 2179.796,E2 2179.796} C_VEL
LIN {X 0,Y 242.675,Z 686.623,A -85,B 0,C 180,E1 2179.496,E2 2179.496} C_VEL
LIN {X 0,Y 242.715,Z 686.599,A -85,B 0,C 180,E1 2174.504,E2 2174.504} C_VEL
LIN {X 0,Y 243.077,Z 688.434,A -85,B 0,C 180,E1 2171.771,E2 2171.771} C_VEL
LIN {X 0,Y 235.794,Z 740.93,A -85,B 0,C 180,E1 2171.222,E2 2171.222} C_VEL
LIN {X 0,Y 230.807,Z 763.252,A -85,B 0,C 180,E1 2170.997,E2 2170.997} C_VEL
LIN {X 0,Y 224.222,Z 784.379,A -85,B 0,C 180,E1 2170.823,E2 2170.823} C_VEL
LIN {X 0,Y 215.989,Z 805.029,A -85,B 0,C 180,E1 2170.601,E2 2170.601} C_VEL
LIN {X 0,Y 205.931,Z 825.453,A -85,B 0,C 180,E1 2170.275,E2 2170.275} C_VEL
LIN {X 0,Y 194.864,Z 844.149,A -85,B 0,C 180,E1 2169.856,E2 2169.856} C_VEL
LIN {X 0,Y 181.87,Z 862.588,A -85,B 0,C 180,E1 2169.28,E2 2169.28} C_VEL
LIN {X 0,Y 167.855,Z 879.429,A -85,B 0,C 180,E1 2168.544,E2 2168.544} C_VEL
LIN {X 0,Y 152.295,Z 895.455,A -85,B 0,C 180,E1 2167.546,E2 2167.546} C_VEL
LIN {X 0,Y 135.797,Z 910.018,A -85,B 0,C 180,E1 2166.22,E2 2166.22} C_VEL
LIN {X 0,Y 118.351,Z 923.198,A -85,B 0,C 180,E1 2164.406,E2 2164.406} C_VEL
LIN {X 0,Y 99.549,Z 935.195,A -85,B 0,C 180,E1 2161.728,E2 2161.728} C_VEL
LIN {X 0,Y 81.063,Z 945.062,A -85,B 0,C 180,E1 2157.871,E2 2157.871} C_VEL
LIN {X 0,Y 62.665,Z 953.299,A -85,B 0,C 180,E1 2151.711,E2 2151.711} C_VEL
LIN {X 0,Y 44.954,Z 959.967,A -85,B 0,C 180,E1 2140.515,E2 2140.515} C_VEL
LIN {X 0,Y 30.761,Z 964.771,A -85,B 0,C 180,E1 2118.439,E2 2118.439} C_VEL
LIN {X 0,Y 25.122,Z 967.696,A -85,B 0,C 180,E1 2081.528,E2 2081.528} C_VEL
LIN {X 0,Y 25.471,Z 968.267,A -85,B 0,C 180,E1 2070.048,E2 2070.048} C_VEL
LIN {X 0,Y 27.652,Z 968.816,A -85,B 0,C 180,E1 2032.127,E2 2032.127} C_VEL
LIN {X 0,Y 42.083,Z 967.939,A -85,B 0,C 180,E1 2002.168,E2 2002.168} C_VEL
LIN {X 0,Y 57.979,Z 966.129,A -85,B 0,C 180,E1 1990.587,E2 1990.587} C_VEL
LIN {X 0,Y 56.416,Z 966.206,A -85,B 0,C 180,E1 1989.908,E2 1989.908} C_VEL
LIN {X 0,Y 48.632,Z 966.839,A -85,B 0,C 180,E1 1990.831,E2 1990.831} C_VEL
LIN {X 0,Y 32.229,Z 967.807,A -85,B 0,C 180,E1 1999.227,E2 1999.227} C_VEL
LIN {X 0,Y 24.849,Z 967.944,A -85,B 0,C 180,E1 2010.025,E2 2010.025} C_VEL
LIN {X 0,Y 17.2,Z 967.503,A -85,B 0,C 180,E1 2063.395,E2 2063.395} C_VEL
LIN {X 0,Y 17.279,Z 967.239,A -85,B 0,C 180,E1 2073.388,E2 2073.388} C_VEL
LIN {X 0,Y 21.867,Z 964.88,A -85,B 0,C 180,E1 2121.103,E2 2121.103} C_VEL
LIN {X 0,Y 37.923,Z 960.251,A -85,B 0,C 180,E1 2147.438,E2 2147.438} C_VEL
LIN {X 0,Y 57.055,Z 953.815,A -85,B 0,C 180,E1 2157.764,E2 2157.764} C_VEL
LIN {X 0,Y 76.102,Z 945.925,A -85,B 0,C 180,E1 2162.847,E2 2162.847} C_VEL
LIN {X 0,Y 95.706,Z 935.917,A -85,B 0,C 180,E1 2165.999,E2 2165.999} C_VEL
LIN {X 0,Y 114.109,Z 924.651,A -85,B 0,C 180,E1 2167.987,E2 2167.987} C_VEL
LIN {X 0,Y 131.762,Z 911.899,A -85,B 0,C 180,E1 2169.384,E2 2169.384} C_VEL
LIN {X 0,Y 148.432,Z 897.785,A -85,B 0,C 180,E1 2170.394,E2 2170.394} C_VEL
LIN {X 0,Y 164.09,Z 882.262,A -85,B 0,C 180,E1 2171.149,E2 2171.149} C_VEL
LIN {X 0,Y 178.711,Z 865.201,A -85,B 0,C 180,E1 2171.711,E2 2171.711} C_VEL
LIN {X 0,Y 191.774,Z 847.291,A -85,B 0,C 180,E1 2172.135,E2 2172.135} C_VEL
LIN {X 0,Y 203.878,Z 827.601,A -85,B 0,C 180,E1 2172.462,E2 2172.462} C_VEL
LIN {X 0,Y 213.929,Z 807.931,A -85,B 0,C 180,E1 2172.69,E2 2172.69} C_VEL
LIN {X 0,Y 222.556,Z 787.192,A -85,B 0,C 180,E1 2172.848,E2 2172.848} C_VEL
LIN {X 0,Y 229.684,Z 765.001,A -85,B 0,C 180,E1 2172.968,E2 2172.968} C_VEL
LIN {X 0,Y 234.716,Z 743.413,A -85,B 0,C 180,E1 2173.14,E2 2173.14} C_VEL
LIN {X 0,Y 239.305,Z 713.068,A -85,B 0,C 180,E1 2173.427,E2 2173.427} C_VEL
LIN {X 0,Y 241.718,Z 695.007,A -85,B 0,C 180,E1 2173.638,E2 2173.638} C_VEL
LIN {X 0,Y 241.487,Z 694.318,A -85,B 0,C 180,E1 2176.106,E2 2176.106} C_VEL
LIN {X 0,Y 241.458,Z 694.498,A -85,B 0,C 180,E1 2177.708,E2 2177.708} C_VEL
LIN {X 0,Y 234.961,Z 739.872,A -85,B 0,C 180,E1 2178.081,E2 2178.081} C_VEL
LIN {X 0,Y 229.853,Z 762.355,A -85,B 0,C 180,E1 2178.296,E2 2178.296} C_VEL
LIN {X 0,Y 223.024,Z 783.925,A -85,B 0,C 180,E1 2178.561,E2 2178.561} C_VEL
LIN {X 0,Y 215.049,Z 803.637,A -85,B 0,C 180,E1 2178.874,E2 2178.874} C_VEL
LIN {X 0,Y 204.99,Z 823.866,A -85,B 0,C 180,E1 2179.285,E2 2179.285} C_VEL
LIN {X 0,Y 193.913,Z 842.39,A -85,B 0,C 180,E1 2179.765,E2 2179.765} C_VEL
LIN {X 0,Y 180.974,Z 860.599,A -85,B 0,C 180,E1 2180.37,E2 2180.37} C_VEL
LIN {X 0,Y 167.2,Z 876.975,A -85,B 0,C 180,E1 2181.096,E2 2181.096} C_VEL
LIN {X 0,Y 152.06,Z 892.425,A -85,B 0,C 180,E1 2182.013,E2 2182.013} C_VEL
LIN {X 0,Y 135.97,Z 906.517,A -85,B 0,C 180,E1 2183.174,E2 2183.174} C_VEL
LIN {X 0,Y 118.875,Z 919.326,A -85,B 0,C 180,E1 2184.696,E2 2184.696} C_VEL
LIN {X 0,Y 100.821,Z 930.686,A -85,B 0,C 180,E1 2186.782,E2 2186.782} C_VEL
LIN {X 0,Y 81.868,Z 940.685,A -85,B 0,C 180,E1 2189.847,E2 2189.847} C_VEL
LIN {X 0,Y 62.151,Z 949.242,A -85,B 0,C 180,E1 2194.837,E2 2194.837} C_VEL
LIN {X 0,Y 43.588,Z 955.801,A -85,B 0,C 180,E1 2203.49,E2 2203.49} C_VEL
LIN {X 0,Y 26.6,Z 960.76,A -85,B 0,C 180,E1 2223.137,E2 2223.137} C_VEL
LIN {X 0,Y 17.977,Z 963.676,A -85,B 0,C 180,E1 2262.784,E2 2262.784} C_VEL
LIN {X 0,Y 19.851,Z 965.369,A -85,B 0,C 180,E1 2306.345,E2 2306.345} C_VEL
LIN {X 0,Y 33.973,Z 966.8,A -85,B 0,C 180,E1 2340.233,E2 2340.233} C_VEL
LIN {X 0,Y 43.448,Z 966.964,A -85,B 0,C 180,E1 2348.499,E2 2348.499} C_VEL
LIN {X 0,Y 24.849,Z 967.944,A -85,B 0,C 180,E1 2370.025,E2 2370.025} C_VEL
LIN {X 0,Y 20.301,Z 967.866,A -85,B 0,C 180,E1 2379.711,E2 2379.711} C_VEL
LIN {X 0,Y 13.699,Z 967.309,A -85,B 0,C 180,E1 2396.947,E2 2396.947} C_VEL
LIN {X 0,Y 9.197,Z 966.182,A -85,B 0,C 180,E1 2443.608,E2 2443.608} C_VEL
LIN {X 0,Y 21.481,Z 963.006,A -85,B 0,C 180,E1 2508.077,E2 2508.077} C_VEL
LIN {X 0,Y 41.033,Z 957.927,A -85,B 0,C 180,E1 2521.75,E2 2521.75} C_VEL
LIN {X 0,Y 61.457,Z 950.884,A -85,B 0,C 180,E1 2526.91,E2 2526.91} C_VEL
LIN {X 0,Y 81.132,Z 942.323,A -85,B 0,C 180,E1 2529.551,E2 2529.551} C_VEL
LIN {X 0,Y 100.938,Z 931.791,A -85,B 0,C 180,E1 2531.234,E2 2531.234} C_VEL
LIN {X 0,Y 118.724,Z 920.503,A -85,B 0,C 180,E1 2532.295,E2 2532.295} C_VEL
LIN {X 0,Y 136.872,Z 906.84,A -85,B 0,C 180,E1 2533.09,E2 2533.09} C_VEL
LIN {X 0,Y 153.329,Z 892.163,A -85,B 0,C 180,E1 2533.654,E2 2533.654} C_VEL
LIN {X 0,Y 168.7,Z 876.141,A -85,B 0,C 180,E1 2534.065,E2 2534.065} C_VEL
LIN {X 0,Y 183.233,Z 858.344,A -85,B 0,C 180,E1 2534.382,E2 2534.382} C_VEL
LIN {X 0,Y 195.813,Z 840.18,A -85,B 0,C 180,E1 2534.602,E2 2534.602} C_VEL
LIN {X 0,Y 206.811,Z 821.308,A -85,B 0,C 180,E1 2534.759,E2 2534.759} C_VEL
LIN {X 0,Y 216.219,Z 801.684,A -85,B 0,C 180,E1 2534.863,E2 2534.863} C_VEL
LIN {X 0,Y 224.199,Z 781.16,A -85,B 0,C 180,E1 2534.922,E2 2534.922} C_VEL
LIN {X 0,Y 230.773,Z 759.297,A -85,B 0,C 180,E1 2534.99,E2 2534.99} C_VEL
LIN {X 0,Y 235.437,Z 737.76,A -85,B 0,C 180,E1 2535.138,E2 2535.138} C_VEL
LIN {X 0,Y 240.458,Z 702.292,A -85,B 0,C 180,E1 2535.434,E2 2535.434} C_VEL
LIN {X 0,Y 240.414,Z 702.329,A -85,B 0,C 180,E1 2535.865,E2 2535.865} C_VEL
LIN {X 0,Y 234.774,Z 740.813,A -85,B 0,C 180,E1 2536.136,E2 2536.136} C_VEL
LIN {X 0,Y 229.66,Z 763.11,A -85,B 0,C 180,E1 2536.307,E2 2536.307} C_VEL
LIN {X 0,Y 222.826,Z 784.542,A -85,B 0,C 180,E1 2536.511,E2 2536.511} C_VEL
LIN {X 0,Y 214.595,Z 804.719,A -85,B 0,C 180,E1 2536.754,E2 2536.754} C_VEL
LIN {X 0,Y 204.5,Z 824.821,A -85,B 0,C 180,E1 2537.06,E2 2537.06} C_VEL
LIN {X 0,Y 193.351,Z 843.296,A -85,B 0,C 180,E1 2537.414,E2 2537.414} C_VEL
LIN {X 0,Y 180.416,Z 861.375,A -85,B 0,C 180,E1 2537.85,E2 2537.85} C_VEL
LIN {X 0,Y 165.972,Z 878.377,A -85,B 0,C 180,E1 2538.392,E2 2538.392} C_VEL
LIN {X 0,Y 151.253,Z 893.203,A -85,B 0,C 180,E1 2539.019,E2 2539.019} C_VEL
LIN {X 0,Y 135.004,Z 907.289,A -85,B 0,C 180,E1 2539.829,E2 2539.829} C_VEL
LIN {X 0,Y 117.731,Z 920.082,A -85,B 0,C 180,E1 2540.876,E2 2540.876} C_VEL
LIN {X 0,Y 99.435,Z 931.43,A -85,B 0,C 180,E1 2542.29,E2 2542.29} C_VEL
LIN {X 0,Y 80.01,Z 941.473,A -85,B 0,C 180,E1 2544.357,E2 2544.357} C_VEL
LIN {X 0,Y 59.851,Z 949.963,A -85,B 0,C 180,E1 2547.658,E2 2547.658} C_VEL
LIN {X 0,Y 40.722,Z 956.407,A -85,B 0,C 180,E1 2553.352,E2 2553.352} C_VEL
LIN {X 0,Y 22.181,Z 961.252,A -85,B 0,C 180,E1 2567.382,E2 2567.382} C_VEL
LIN {X 0,Y 10.08,Z 964.308,A -85,B 0,C 180,E1 2617.177,E2 2617.177} C_VEL
LIN {X 0,Y 14.344,Z 966.072,A -85,B 0,C 180,E1 2686.998,E2 2686.998} C_VEL
LIN {X 0,Y 24.469,Z 967.098,A -85,B 0,C 180,E1 2708.102,E2 2708.102} C_VEL
LIN {X 0,Y 9.279,Z 966.646,A -85,B 0,C 180,E1 2771.279,E2 2771.279} C_VEL
LIN {X 0,Y 9.338,Z 966.428,A -85,B 0,C 180,E1 2790.131,E2 2790.131} C_VEL
LIN {X 0,Y 9.197,Z 966.182,A -85,B 0,C 180,E1 2803.608,E2 2803.608} C_VEL
LIN {X 0,Y 11.085,Z 965.174,A -85,B 0,C 180,E1 2843.396,E2 2843.396} C_VEL
LIN {X 0,Y 19.192,Z 962.812,A -85,B 0,C 180,E1 2879.201,E2 2879.201} C_VEL
LIN {X 0,Y 29.571,Z 960.067,A -85,B 0,C 180,E1 2891.08,E2 2891.08} C_VEL
LIN {X 0,Y 33.851,Z 958.902,A -85,B 0,C 180,E1 2892.321,E2 2892.321} C_VEL
LIN {X 0,Y 54.644,Z 952.502,A -85,B 0,C 180,E1 2894.038,E2 2894.038} C_VEL
LIN {X 0,Y 74.545,Z 944.62,A -85,B 0,C 180,E1 2894.987,E2 2894.987} C_VEL
LIN {X 0,Y 94.498,Z 934.707,A -85,B 0,C 180,E1 2895.626,E2 2895.626} C_VEL
LIN {X 0,Y 113.429,Z 923.325,A -85,B 0,C 180,E1 2896.06,E2 2896.06} C_VEL
LIN {X 0,Y 131.322,Z 910.537,A -85,B 0,C 180,E1 2896.368,E2 2896.368} C_VEL
LIN {X 0,Y 134.829,Z 907.782,A -85,B 0,C 180,E1 2896.438,E2 2896.438} C_VEL
LIN {X 0,Y 117.118,Z 920.813,A -85,B 0,C 180,E1 2896.998,E2 2896.998} C_VEL
LIN {X 0,Y 97.65,Z 932.753,A -85,B 0,C 180,E1 2897.744,E2 2897.744} C_VEL
LIN {X 0,Y 78.135,Z 942.613,A -85,B 0,C 180,E1 2898.704,E2 2898.704} C_VEL
LIN {X 0,Y 58.323,Z 950.758,A -85,B 0,C 180,E1 2900.055,E2 2900.055} C_VEL
LIN {X 0,Y 37.844,Z 957.392,A -85,B 0,C 180,E1 2902.294,E2 2902.294} C_VEL
LIN {X 0,Y 18.006,Z 962.195,A -85,B 0,C 180,E1 2907.175,E2 2907.175} C_VEL
LIN {X 0,Y 2.058,Z 965.077,A -85,B 0,C 180,E1 2956.723,E2 2956.723} C_VEL
LIN {X 0,Y 4.124,Z 965.784,A -85,B 0,C 180,E1 3065.762,E2 3065.762} C_VEL
LIN {X 0,Y 1.263,Z 965.434,A -85,B 0,C 180,E1 3175.725,E2 3175.725} C_VEL
LIN {X 0,Y 19.299,Z 962.323,A -85,B 0,C 180,E1 3249.786,E2 3249.786} C_VEL
LIN {X 0,Y 33.851,Z 958.902,A -85,B 0,C 180,E1 3252.321,E2 3252.321} C_VEL
LIN {X 0,Y 36.356,Z 960.835,A -85,B 0,C 180,E1 3252.594,E2 3252.594} C_VEL
LIN {X 0,Y 36.356,Z 1015.5,A -85,B 0,C 180,E1 3252.594,E2 3252.594} C_VEL
LIN {X 0,Y 36.356,Z 1015.5,A -85,B 0,C 180,E1 3252.594,E2 3252.594}

QRS_NEXT_CUT()

QRS_NEXT()
QRS_HOME()

END
